Staubli VAL3: LINESYM.pgx

public program LineSym(trsf x_trSource, trsf& x_trLine[], trsf& x_trDest, bool& x_bRes)
  local frame l_fFrame
  local point l_p
  local trsf l_trT[3]
begin

  //有关直线对称


  l_trT[0]=x_trLine[0]
  l_trT[1]=x_trLine[1]
  l_trT[2]=x_trSource

  call SetFrame(l_trT,l_fFrame,x_bRes)
  if !x_bRes
    return
  endIf

  l_p.trsf=x_trSource
  link(l_p,world)
  l_p.trsf=position(l_p,l_fFrame)
  l_p.trsf.y=-l_p.trsf.y
  link(l_p,l_fFrame)
  x_trDest=position(l_p,world)



end
